{attribute 'GeneratedUsingTerminal: KL3362'}
{attribute addProperty BoxType "KL3362"}
{attribute addProperty Id "Channel_1AT %Q*Channel_3C1A65000Channel_2AT %Q*Channel_3C1A65000"}
{attribute addProperty CRC "3918264561"}
{attribute addProperty Size "0"}
TYPE KL3362_E98BF8F1 :
STRUCT
	{attribute addProperty Name "Channel_1"}
	Channel_1 : Channel_3C1A6500;
	{attribute addProperty Name "Channel_2"}
	Channel_2 : Channel_3C1A6500;
END_STRUCT
END_TYPE

(* stored: Version 1.2.0.0, ProductVersion 3.1.4024.9
   DUT KL3362_E98BF8F1: Id {c1fbb13c-ce65-4b3b-aa59-af45b8c66c02} *)
